FUNCTION_BLOCK KulaMatlyft
  (* Version 0.1, 2005-05-13, MFBL, Chalmers *)
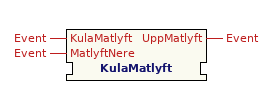
  EVENT_INPUT
    KulaMatlyft;
    MatlyftNere;
  END_EVENT
  EVENT_OUTPUT
    UppMatlyft;
  END_EVENT
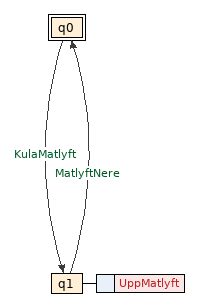
  EC_STATES
    q0;
    q1 : -> UppMatlyft;
  END_STATES
  EC_TRANSITIONS
    q0 TO q1 := KulaMatlyft;
    q1 TO q0 := MatlyftNere;
  END_TRANSITIONS
END_FUNCTION_BLOCK
